(* CODESYS project mobject-graph-api.library
   Company: mobject
   DefaultNamespace: mobject-graph-api
   Version: 0.6.0
   Placeholder: mobject-graph-api
   Author: mobject dev team
   Title: mobject-graph-api

Project tree, tasks and I/O mapping:
  libraries: mobject-collections, 1.3.0 (mobject); mobject-deserialization, 0.3.0 (mobject); mobject-events, 1.1.0 (mobject); mobject-graph, 0.5.0 (mobject); mobject-serialization, 0.5.0 (mobject); mobject-server, 0.6.0 (mobject); Tc2_Standard, * (Beckhoff Automation GmbH); Tc2_System, * (Beckhoff Automation GmbH)
  _Internal/
    Handlers/
      function block CreateGraphMultiUserRpcHandler [ST]: Handle, Initialize
      function block CreateGraphRpcHandler [ST]: Handle, Initialize
      function block GetBlueprintsRpcHandler [ST]: Handle, Initialize
      function block GetContentValueHandler [ST]: Handle, Initialize
      function block GetStatusRpcHandler [ST]: Handle, Initialize
    Visitors/
      function block GetBlueprintsVisitor [ST]: Initialize, VisitAlarm, VisitContent, VisitExtension, VisitInputPort, VisitMetadatum, VisitNode, VisitNodeFactory, VisitNodePrototype, VisitOutputPort, VisitParameter
      function block RetrieveNodeContentValue [ST]: LogInvalidContentNameError, LogInvalidNodeIdError, Reset, Done, Error, ErrorMessage, Initialize, VisitContent, VisitGraph, VisitNode
  function block GraphApi [ST]: FB_init, FB_exit, Graphs, OffEvent, OnceEvent, OnEvent, RegisterWith
*)

// _Internal/Handlers/CreateGraphMultiUserRpcHandler
{attribute 'linkalways'} 
{attribute 'no_explicit_call' := 'This FB is a CLASS and must be accessed using methods or properties'}
{attribute 'enable_dynamic_creation'}
FUNCTION_BLOCK CreateGraphMultiUserRpcHandler IMPLEMENTS I_RpcHandler
VAR
	graphFramework : I_GraphFramework;
	graphs : I_Graphs;
	userGraphs : Dictionary;
END_VAR

METHOD Handle
VAR_INPUT
	Parameters : I_Deserializer;
	Response : I_SynchronousRpcResponse;
END_VAR
VAR
	clientId : T_MAXSTRING;
	graphUuid : T_MAXSTRING;
	graph : I_Graph;
	feedback : DeserializerFeedback;
	graphDeserializer : I_Deserializer;
END_VAR
IF NOT Parameters.TryGetKeyString('clienId', clientId, feedback) THEN
	Response.RejectWithMessage(feedback.FirstError.Message);
	RETURN;
END_IF

IF NOT userGraphs.TryGetValue(clientId, graphUuid) THEN
	IF graphs.TryGetGraphByUuid(graphUuid,graph) THEN
		graphs.RemoveGraph(graph);
		graph.Dispose();
	END_IF
	userGraphs.Remove(clientId);
END_IF

graph := graphFramework.Create();
graphDeserializer := Parameters.GetKeyObject('graph');

IF NOT graph.TryDeserializeFrom(graphDeserializer, feedback) THEN
	Response.RejectWithMessage(feedback.FirstError.Message);
	graph.Dispose();
	RETURN;
END_IF

graphUuid := graph.Uuid;
userGraphs.AddOrUpdate(clientId, graphUuid);
graphs.AddGraph(graph);
Response.CompleteWithObject(graph);
END_METHOD

METHOD PUBLIC Initialize
VAR_INPUT
	GraphFramework : I_GraphFramework;
	Graphs : I_Graphs;
END_VAR
THIS^.graphFramework := GraphFramework;
THIS^.graphs := Graphs;
END_METHOD

END_FUNCTION_BLOCK

// _Internal/Handlers/CreateGraphRpcHandler
{attribute 'linkalways'} 
{attribute 'no_explicit_call' := 'This FB is a CLASS and must be accessed using methods or properties'}
{attribute 'enable_dynamic_creation'}
FUNCTION_BLOCK CreateGraphRpcHandler IMPLEMENTS I_RpcHandler
VAR
	graphFramework : I_GraphFramework;
	graphs : I_Graphs;
	lastGraphUuid : T_MAXSTRING;
END_VAR

METHOD Handle
VAR_INPUT
	Parameters : I_Deserializer;
	Response : I_SynchronousRpcResponse;
END_VAR
VAR
	graph : I_Graph;
	feedback : DeserializerFeedback;
	graphDeserializer : I_Deserializer;
END_VAR
IF graphs.TryGetGraphByUuid(lastGraphUuid,graph) THEN
	graphs.RemoveGraph(graph);
	graph.Dispose();
	lastGraphUuid := '';
END_IF

graph := graphFramework.Create();
graphDeserializer := Parameters.GetKeyObject('graph');

IF NOT graph.TryDeserializeFrom(graphDeserializer, feedback) THEN
	Response.RejectWithMessage(feedback.FirstError.Message);
	graph.Dispose();
	RETURN;
END_IF

lastGraphUuid := graph.Uuid;
graphs.AddGraph(graph);
Response.CompleteWithObject(graph);
END_METHOD

METHOD PUBLIC Initialize
VAR_INPUT
	GraphFramework : I_GraphFramework;
	Graphs : I_Graphs;
END_VAR
THIS^.graphFramework := GraphFramework;
THIS^.graphs := Graphs;
END_METHOD

END_FUNCTION_BLOCK

// _Internal/Handlers/GetBlueprintsRpcHandler
{attribute 'linkalways'} 
{attribute 'no_explicit_call' := 'This FB is a CLASS and must be accessed using methods or properties'}
{attribute 'enable_dynamic_creation'}
FUNCTION_BLOCK GetBlueprintsRpcHandler IMPLEMENTS I_RpcHandler
VAR
	nodeFactory : I_NodeFactory;
END_VAR

METHOD Handle
VAR_INPUT
	Parameters : I_Deserializer;
	Response : I_SynchronousRpcResponse;
END_VAR
VAR
	visitor : GetBlueprintsVisitor;
	serializer : I_Serializer;
END_VAR
IF nodeFactory = 0 THEN
	Response.RejectWithMessage('GetBlueprintsRpcHandler has not been initialized with a valid nodeFactory object');
	RETURN;
END_IF

serializer := Response.GetSerializer();
visitor.Initialize(serializer);
nodeFactory.Accept(visitor);

Response.CompleteWithSerializer(serializer);
serializer.Dispose();
END_METHOD

METHOD PUBLIC Initialize
VAR_INPUT
	NodeFactory : I_NodeFactory;
END_VAR
this^.nodeFactory := NodeFactory;
END_METHOD

END_FUNCTION_BLOCK

// _Internal/Visitors/GetBlueprintsVisitor
{attribute 'linkalways'} 
{attribute 'no_explicit_call' := 'This FB is a CLASS and must be accessed using methods or properties'}
{attribute 'enable_dynamic_creation'}
FUNCTION_BLOCK GetBlueprintsVisitor IMPLEMENTS I_NodeFactoryVisitor, I_NodePrototypeVisitor, I_NodeVisitor, I_ExtensionVisitor, I_InputPortVisitor, I_OutputPortVisitor, I_MetadataVisitor, I_ContentVisitor, I_ParameterVisitor, I_AlarmVisitor
VAR
	serializer : I_Serializer;
END_VAR

METHOD PUBLIC Initialize
VAR_INPUT
	Serializer : I_Serializer;
END_VAR
THIS^.serializer := Serializer;
END_METHOD

METHOD VisitAlarm
VAR_INPUT
	VisitingAlarm : I_Alarm;
END_VAR
serializer.AddString(VisitingAlarm.Message);
END_METHOD

METHOD VisitContent
VAR_INPUT
	VisitingContent : I_Content;
END_VAR
serializer.StartObject();

serializer.AddKeyString('name',VisitingContent.Name);
serializer.Addkey('datatype');
VisitingContent.Data.SerializeTypeWith(serializer);

IF VisitingContent.Metadatum.HasMetadata THEN
	serializer.addkey('metadata');
	serializer.StartArray();
	VisitingContent.Metadatum.Accept(THIS^);
	serializer.EndArray();
END_IF

serializer.EndObject();
END_METHOD

METHOD VisitExtension
VAR_INPUT
	VisitingExtension : I_Extension;
END_VAR
Serializer.StartObject();
Serializer.AddKeyString('name',VisitingExtension.Name);

IF VisitingExtension.Metadatum.HasMetadata THEN
	serializer.addkey('metadata');
	serializer.StartArray();
	VisitingExtension.Metadatum.Accept(THIS^);
	serializer.EndArray();
END_IF

IF VisitingExtension.Alarms.HasAlarms THEN
	serializer.addkey('alarms');
	serializer.StartArray();
	VisitingExtension.Alarms.Accept(THIS^);
	serializer.EndArray();
END_IF

IF VisitingExtension.InputPorts.HasInputPorts THEN
	serializer.addkey('inputPorts');
	serializer.StartArray();
	VisitingExtension.InputPorts.Accept(THIS^);
	serializer.EndArray();
END_IF

IF VisitingExtension.OutputPorts.HasOutputPorts THEN
	serializer.addkey('outputPorts');
	serializer.StartArray();
	VisitingExtension.OutputPorts.Accept(THIS^);
	serializer.EndArray();
END_IF

IF VisitingExtension.Parameters.HasParameters THEN
	serializer.addkey('parameters');
	serializer.StartArray();
	VisitingExtension.Parameters.Accept(THIS^);
	serializer.EndArray();
END_IF

IF VisitingExtension.Contents.HasContents THEN
	serializer.addkey('contents');
	serializer.StartArray();
	VisitingExtension.Parameters.Accept(THIS^);
	serializer.EndArray();
END_IF

Serializer.EndObject();
END_METHOD

METHOD VisitInputPort
VAR_INPUT
	VisitingInputPort : I_InputPort;
END_VAR
serializer.StartObject();

serializer.AddKeyString('name',VisitingInputPort.Name);
serializer.Addkey('datatype');
VisitingInputPort.Data.SerializeTypeWith(serializer);

IF VisitingInputPort.Metadatum.HasMetadata THEN
	serializer.addkey('metadata');
	serializer.StartArray();
	VisitingInputPort.Metadatum.Accept(THIS^);
	serializer.EndArray();
END_IF

serializer.EndObject();
END_METHOD

METHOD VisitMetadatum
VAR_INPUT
	VisitingMetadatum : I_Metadata;
END_VAR
serializer.StartObject();
serializer.AddKeyString('name',VisitingMetadatum.Name);
serializer.AddkeyObject('value',VisitingMetadatum.Data);
serializer.EndObject();
END_METHOD

METHOD VisitNode
VAR_INPUT
	VisitingNode : I_Node;
END_VAR
serializer.StartObject();

IF VisitingNode.Metadatum.HasMetadata THEN
	serializer.addkey('metadata');
	serializer.StartArray();
	VisitingNode.Metadatum.Accept(THIS^);
	serializer.EndArray();
END_IF

IF VisitingNode.Alarms.HasAlarms THEN
	serializer.addkey('alarms');
	serializer.StartArray();
	VisitingNode.Alarms.Accept(THIS^);
	serializer.EndArray();
END_IF

IF VisitingNode.Extensions.HasExtensions THEN
	serializer.addkey('extensions');
	serializer.StartArray();
	VisitingNode.Extensions.Accept(THIS^);
	serializer.EndArray();
END_IF

IF VisitingNode.InputPorts.HasInputPorts THEN
	serializer.addkey('inputPorts');
	serializer.StartArray();
	VisitingNode.InputPorts.Accept(THIS^);
	serializer.EndArray();
END_IF

IF VisitingNode.OutputPorts.HasOutputPorts THEN
	serializer.addkey('outputPorts');
	serializer.StartArray();
	VisitingNode.OutputPorts.Accept(THIS^);
	serializer.EndArray();
END_IF

IF VisitingNode.Parameters.HasParameters THEN
	serializer.addkey('parameters');
	serializer.StartArray();
	VisitingNode.Parameters.Accept(THIS^);
	serializer.EndArray();
END_IF

IF VisitingNode.Contents.HasContents THEN
	serializer.addkey('contents');
	serializer.StartArray();
	VisitingNode.Contents.Accept(THIS^);
	serializer.EndArray();
END_IF

serializer.EndObject();
END_METHOD

METHOD VisitNodeFactory
VAR_INPUT
	VisitingNodeFactory : I_NodeFactory;
END_VAR
serializer.StartObject();
serializer.AddKey('blueprints');
serializer.StartArray();
VisitingNodeFactory.NodePrototypes.Accept(THIS^);
serializer.EndArray();
serializer.EndObject();
END_METHOD

METHOD VisitNodePrototype
VAR_INPUT
	VisitingPrototype : I_NodePrototype;
END_VAR
serializer.StartObject();
serializer.AddKeyString('path',VisitingPrototype.Path);
serializer.AddKey('node');
VisitingPrototype.Node.Accept(THIS^);
serializer.EndObject();
END_METHOD

METHOD VisitOutputPort
VAR_INPUT
	VisitingOutputPort : I_OutputPort;
END_VAR
serializer.StartObject();

serializer.AddKeyString('name',VisitingOutputPort.Name);
serializer.Addkey('datatype');
VisitingOutputPort.Data.SerializeTypeWith(serializer);

IF VisitingOutputPort.Metadatum.HasMetadata THEN
	serializer.addkey('metadata');
	serializer.StartArray();
	VisitingOutputPort.Metadatum.Accept(THIS^);
	serializer.EndArray();
END_IF

serializer.EndObject();
END_METHOD

METHOD VisitParameter
VAR_INPUT
	VisitingProperty : I_Parameter;
END_VAR
serializer.StartObject();

serializer.AddKeyString('name',VisitingProperty.Name);
serializer.Addkey('datatype');
VisitingProperty.Data.SerializeTypeWith(serializer);
serializer.Addkey('defaultValue');
VisitingProperty.Data.SerializeWith(serializer);

IF VisitingProperty.Metadatum.HasMetadata THEN
	serializer.addkey('metadata');
	serializer.StartArray();
	VisitingProperty.Metadatum.Accept(THIS^);
	serializer.EndArray();
END_IF

Serializer.EndObject();
END_METHOD

END_FUNCTION_BLOCK

// _Internal/Handlers/GetContentValueHandler
{attribute 'linkalways'} 
{attribute 'no_explicit_call' := 'This FB is a CLASS and must be accessed using methods or properties'}
{attribute 'enable_dynamic_creation'}
FUNCTION_BLOCK GetContentValueHandler IMPLEMENTS I_RpcHandler
VAR
	graphs : I_Graphs;
END_VAR

METHOD Handle
VAR_INPUT
	Parameters : I_Deserializer;
	Response : I_SynchronousRpcResponse;
END_VAR
VAR
	graphUuid : T_MAXSTRING;
	nodeId : T_MAXSTRING;
	contentName : T_MAXSTRING;
	visitor : RetrieveNodeContentValue;
	serializer : I_Serializer;
	feedback : DeserializerFeedback;
END_VAR
IF NOT Parameters.TryGetKeyString('graphUuid', graphUuid, feedback) THEN
	Response.RejectWithMessage(feedback.FirstError.Message);
	RETURN;
END_IF

IF NOT Parameters.TryGetKeyString('nodeId', nodeId, feedback) THEN
	Response.RejectWithMessage(feedback.FirstError.Message);
	RETURN;
END_IF

IF NOT Parameters.TryGetKeyString('contentName', contentName, feedback) THEN
	Response.RejectWithMessage(feedback.FirstError.Message);
	RETURN;
END_IF

serializer := Response.GetSerializer();
visitor.Initialize(graphUuid, nodeId, contentName, serializer);
graphs.Accept(visitor);

IF visitor.Error THEN
	Response.RejectWithMessage(visitor.ErrorMessage);
	serializer.Dispose();
	RETURN;
END_IF

IF NOT visitor.Done THEN
	Response.RejectWithMessage('Invalid graphUuid');
	serializer.Dispose();
	RETURN;
END_IF

Response.CompleteWithSerializer(serializer);
serializer.Dispose();
END_METHOD

METHOD PUBLIC Initialize
VAR_INPUT
	Graphs : I_Graphs;
END_VAR
this^.graphs := Graphs;
END_METHOD

END_FUNCTION_BLOCK

// _Internal/Visitors/RetrieveNodeContentValue
{attribute 'linkalways'} 
{attribute 'no_explicit_call' := 'This FB is a CLASS and must be accessed using methods or properties'}
{attribute 'enable_dynamic_creation'}
FUNCTION_BLOCK RetrieveNodeContentValue IMPLEMENTS I_GraphVisitor, I_NodeVisitor, I_ContentVisitor
VAR
	graphUuid : T_MAXSTRING;
	nodeId : T_MAXSTRING;
	contentName : T_MAXSTRING;
	serializer : I_Serializer;
	_done : BOOL;
	_error : BOOL;
	_errorMessage : T_MAXSTRING;
END_VAR

METHOD PRIVATE LogInvalidContentNameError
VAR_INPUT
END_VAR
_errorMessage := 'Invalid Content Name';
_error := TRUE;
END_METHOD

METHOD PRIVATE LogInvalidNodeIdError
VAR_INPUT
END_VAR
_errorMessage := 'Invalid Node Id';
_error := TRUE;
END_METHOD

METHOD PRIVATE Reset
VAR_INPUT
END_VAR
_done := FALSE;
_errorMessage := '';
_error := FALSE;
END_METHOD

PROPERTY PUBLIC Done : BOOL
GET
Done := _done;
END_GET
END_PROPERTY

PROPERTY PUBLIC Error : BOOL
GET
Error := _error;
END_GET
END_PROPERTY

PROPERTY PUBLIC ErrorMessage : T_MAXSTRING
GET
ErrorMessage := _errorMessage;
END_GET
END_PROPERTY

METHOD PUBLIC Initialize
VAR_INPUT
	GraphUuid : T_MAXSTRING;
	NodeId : T_MAXSTRING;
	ContentName : T_MAXSTRING;
	Serializer : I_Serializer;
END_VAR
THIS^.graphUuid := GraphUuid;
THIS^.nodeId := NodeId;
THIS^.contentName := ContentName;
THIS^.serializer := Serializer;
END_METHOD

METHOD VisitContent
VAR_INPUT
	VisitingContent : I_Content;
END_VAR
VisitingContent.SerializeWith(serializer);
END_METHOD

METHOD VisitGraph
VAR_INPUT
	VisitingGraph : I_Graph;
END_VAR
VAR
	node : I_Node;
END_VAR
Reset();

IF NOT (VisitingGraph.Uuid = graphUuid) THEN
	RETURN;
END_IF

IF NOT VisitingGraph.Nodes.TryGetNodeById(nodeId, node) THEN
	LogInvalidNodeIdError();
	RETURN;
END_IF

node.Accept(THIS^);
END_METHOD

METHOD VisitNode
VAR_INPUT
	VisitingNode : I_Node;
END_VAR
VAR
	content : I_Content;
END_VAR
IF NOT VisitingNode.Contents.TryGetContentByName(contentName, content) THEN
	LogInvalidContentNameError();
	RETURN;
END_IF

content.Accept(THIS^);
END_METHOD

END_FUNCTION_BLOCK

// _Internal/Handlers/GetStatusRpcHandler
{attribute 'linkalways'} 
{attribute 'no_explicit_call' := 'This FB is a CLASS and must be accessed using methods or properties'}
{attribute 'enable_dynamic_creation'}
FUNCTION_BLOCK GetStatusRpcHandler IMPLEMENTS I_RpcHandler
VAR
	graphs : I_Graphs;
END_VAR

METHOD Handle
VAR_INPUT
	Parameters : I_Deserializer;
	Response : I_SynchronousRpcResponse;
END_VAR
VAR
	graphUuid : T_MAXSTRING;
	graph : I_Graph;
	feedback : DeserializerFeedback;
	serializer : I_Serializer;
END_VAR
IF NOT Parameters.TryGetKeyString('graphUuid', graphUuid, feedback) THEN
	Response.RejectWithMessage(feedback.FirstError.Message);
	RETURN;
END_IF

IF NOT graphs.TryGetGraphByUuid(graphUuid,graph) THEN
	Response.RejectWithMessage(concat('Unknown UUID : ',graphUuid));
	RETURN;
END_IF

serializer := Response.GetSerializer();
graph.SerializeWith(serializer);
Response.CompleteWithObject(graph);
serializer.Dispose();
END_METHOD

METHOD PUBLIC Initialize
VAR_INPUT
	Graphs : I_Graphs;
END_VAR
THIS^.graphs := Graphs;
END_METHOD

END_FUNCTION_BLOCK

// GraphApi
{attribute 'linkalways'} 
{attribute 'no_explicit_call' := 'This FB is a CLASS and must be accessed using methods or properties'}
{attribute 'enable_dynamic_creation'}
FUNCTION_BLOCK GraphApi IMPLEMENTS I_RpcApi, I_HostGraphs, I_EventEmitter
VAR
	graphFramework : I_GraphFramework;
	eventEmitter : EventEmitter;
	graphHost : GraphHost(THIS^, eventEmitter);
	createGraphRpcHandler : CreateGraphRpcHandler;
	createGraphMultiUserRpcHandler : CreateGraphMultiUserRpcHandler;
	getStatusRpcHandler : GetStatusRpcHandler;
	getBlueprintsRpcHandler : GetBlueprintsRpcHandler;
	getContentValueHandler : GetContentValueHandler;
END_VAR

METHOD FB_init : BOOL
VAR_INPUT
	bInitRetains : BOOL; // if TRUE, the retain variables are initialized (warm start / cold start)
	bInCopyCode : BOOL;  // if TRUE, the instance afterwards gets moved into the copy code (online change)
	GraphFramework : I_GraphFramework;
END_VAR
THIS^.graphFramework := GraphFramework;
getBlueprintsRpcHandler.Initialize(GraphFramework.NodeFactory);
getStatusRpcHandler.Initialize(graphHost);
createGraphRpcHandler.Initialize(GraphFramework, graphHost);
createGraphMultiUserRpcHandler.Initialize(GraphFramework, graphHost);
getContentValueHandler.Initialize(graphHost);
END_METHOD

METHOD FB_exit : BOOL
VAR_INPUT
	bInCopyCode : BOOL; // if TRUE, the exit method is called for exiting an instance that is copied afterwards (online change).
END_VAR
IF bInCopyCode THEN
	RETURN;
END_IF

graphs.DisposeAll();
END_METHOD

PROPERTY PUBLIC Graphs : I_Graphs
GET
Graphs := graphHost;
END_GET
END_PROPERTY

METHOD PUBLIC OffEvent
VAR_INPUT
	EventName : T_MaxString;
	EventHandler : I_EventHandler;
END_VAR
eventEmitter.OffEvent(EventName, EventHandler);
END_METHOD

METHOD PUBLIC OnceEvent
VAR_INPUT
	EventName : T_MaxString;
	EventHandler : I_EventHandler;
END_VAR
eventEmitter.OnceEvent(EventName, EventHandler);
END_METHOD

METHOD PUBLIC OnEvent
VAR_INPUT
	EventName : T_MaxString;
	EventHandler : I_EventHandler;
END_VAR
eventEmitter.OnEvent(EventName, EventHandler);
END_METHOD

METHOD RegisterWith
VAR_INPUT
	Server : I_RpcServer;
END_VAR
Server.RegisterRpcHandler('CreateGraph',createGraphRpcHandler);
Server.RegisterRpcHandler('CreateGraphMultiUser',createGraphMultiUserRpcHandler);
Server.RegisterRpcHandler('GetStatus',getStatusRpcHandler);
Server.RegisterRpcHandler('GetBlueprints',getBlueprintsRpcHandler);
Server.RegisterRpcHandler('GetContentValue',getContentValueHandler);
END_METHOD

END_FUNCTION_BLOCK
